// TIA Portal V18 export
VAR_GLOBAL   // PLC tag table "AQ"
   outa_BaseAxis AT %QW3 : Int;
   outa_Arm1Axis AT %QW6 : Int;
   outa_Arm2Axis AT %QW8 : Int;
   outa_Arm3Axis AT %QW10 : Int;
   outa_ToolAxis AT %QW12 : Int;
   outa_BaseSpeed AT %QW14 : Int;
   outa_Arm1Speed AT %QW16 : Int;
   outa_Arm2Speed AT %QW18 : Int;
   outa_Arm3Speed AT %QW20 : Int;
   outa_ToolSpeed AT %QW22 : Int;
   outa_10 AT %QW24 : Int;
   outa_11 AT %QW26 : Int;
   outa_HorizontalAxis AT %QW30 : Int;
   outa_VerticalAxis AT %QW32 : Int;
END_VAR
